PROGRAM EtherCAT_Diagnostic
VAR
END_VAR

END_PROGRAM

(* stored: Version 1.1.0.1, ProductVersion 3.1.4024.0
   POU EtherCAT_Diagnostic: Id {a1ab0ab1-8b2f-4cab-a848-d78f1962c48c}, SpecialFunc None *)
